// A timer that triggers at regular intervals. It tracks elapsed time in
// nanoseconds and invokes a user-defined callback when each interval is reached.
// This block is particularly useful in scenarios where repeated actions are
// needed at precise time intervals, such as generating periodic events or
// monitoring cyclic processes.
//
// [usage] 
// The timer can be started with the `Start` method, and the `Run` method should
// be called within a cyclic task to continuously update the timer state. The
// `IntervalCount` property can be used to specify the duration between triggers, and
// the callback method will be called each time this duration is met.
{attribute 'enable_dynamic_creation'}
{attribute 'no_explicit_call' := 'direct call for this function block is not allowed'}
FUNCTION_BLOCK FINAL FB_IntervalTimer IMPLEMENTS I_IntervalTimer
VAR
	_tIntervalTime	: LTIME; // Duration between each interval trigger.
	_tTick			: LTIME; // Timestamp at which the timer was last started or reset.
	_tElapsedTime 	: LTIME; // Total elapsed time since the timer was started.
	_bIsRunning 	: BOOL;  // Indicating whether the interval timer is currently running.
	_IntervalCount 	: FsCommon.T_Size; // Number of intervals that have passed since the timer started.
	_ipCallback 	: I_TimeElapsedCallback; // Reference to the callback that will be invoked when the interval is reached.
END_VAR

// The elapsed time since the timer was started or last reset, showing how much time has passed within the current interval.
// [get] Returns the elapsed time within the current interval.
PROPERTY ElapsedTime  : LTIME
GET
ElapsedTime := THIS^._tElapsedTime;
END_GET
END_PROPERTY

// The number of intervals that have elapsed since the timer was started or reset.
// [get] Returns the number of elapsed intervals.
PROPERTY IntervalCount : FsCommon.T_Size
GET
IntervalCount := THIS^._IntervalCount;
END_GET
END_PROPERTY

// The interval duration for the timer. It specifies how long the timer should wait between triggers.
// [get] Returns the interval duration.
// [set] Sets the interval duration.
PROPERTY IntervalTime : LTIME
GET
IntervalTime := THIS^._tIntervalTime;
END_GET
SET
THIS^._tIntervalTime := IntervalTime;
END_SET
END_PROPERTY

// Indicates whether the interval timer is currently running.
// [get] Returns TRUE if the timer is running; otherwise, FALSE.
PROPERTY IsRunning  : BOOL
GET
IsRunning := THIS^._bIsRunning;
END_GET
END_PROPERTY

// The method that must be called cyclically to run the interval timer.
METHOD Run : I_IntervalTimer // Reference to the current instance of I_IntervalTimer.
VAR_INPUT
END_VAR
Run := THIS^;

IF NOT THIS^._bIsRunning THEN RETURN; END_IF

THIS^._tElapsedTime := LTIME() - THIS^._tTick;

IF THIS^._tElapsedTime < THIS^._tIntervalTime THEN RETURN; END_IF

THIS^._IntervalCount := THIS^._IntervalCount + 1;
IF THIS^._ipCallback <> 0 THEN THIS^._ipCallback.OnTimeElapsed(THIS^); END_IF
THIS^._tTick := LTIME();
END_METHOD

// Sets the callback to be invoked when the interval has elapsed.
METHOD SetCallback : I_IntervalTimer // Reference to the current instance of I_IntervalTimer.
VAR_INPUT
	// The callback that is invoked when the interval elapses.
    ipCallback : I_TimeElapsedCallback;
END_VAR
THIS^._ipCallback := ipCallback;
END_METHOD

// Starts the interval timer, beginning the measurement of time intervals.
METHOD Start : I_IntervalTimer // Reference to the current instance of I_IntervalTimer.
VAR_INPUT
END_VAR
Start := THIS^;

IF THIS^._bIsRunning THEN RETURN; END_IF

THIS^._tElapsedTime 	:= LTIME#0S;
THIS^._IntervalCount 	:= 0;
THIS^._tTick 			:= LTIME();
THIS^._bIsRunning 		:= TRUE;
END_METHOD

// Stops the interval timer, halting the measurement of time intervals.
METHOD Stop : I_IntervalTimer // Reference to the current instance of I_IntervalTimer.
VAR_INPUT
END_VAR
Stop := THIS^;

THIS^._bIsRunning := FALSE;
END_METHOD

END_FUNCTION_BLOCK

(* stored: Version 1.1.0.1
   POU FB_IntervalTimer: Id {af3fb079-5778-4b48-bb34-eeec842df8e4}, SpecialFunc None
   Property ElapsedTime: Id {35433c27-228f-4407-9c69-cde4956e7847}
   Get Get: Id {6fe03b17-d822-4f1d-90b9-4208c02cf341}
   Property IntervalCount: Id {15b69687-6502-4388-b9de-443da2680d67}
   Get Get: Id {0a8ab87c-3eb8-4c02-a746-f9493f19b0d5}
   Property IntervalTime: Id {656d29bd-0108-4834-bbe4-a498af35f48a}
   Get Get: Id {ee0b9fbd-64cd-4d1f-94b0-d9e191df6555}
   Set Set: Id {7a967827-3bd2-4024-8498-4cd74367d440}
   Property IsRunning: Id {a5f627dc-f9b4-4d00-979a-9f8318a120f2}
   Get Get: Id {c7668642-787b-40a8-bea7-2183d4d39a58}
   Method Run: Id {6499b048-2db3-4a7e-a70d-2a35eeb856b8}
   Method SetCallback: Id {fae41798-9332-4ab0-ac9d-94329a59951d}
   Method Start: Id {fb887e9c-57c9-49f6-acd2-436d81766c2d}
   Method Stop: Id {5fbfddc8-814b-4b36-a095-b00fe837c73d} *)
